// TwinCAT 3 PLC project haptix_beckhoff
// Title: Haptix-Beckhoff
// Company: HaptiX Lab
// Author: Nick Janne
// ProjectVersion: 0.5
// Description: This is a library containing a standardized set of function blocks and tools used in research projects at the HaptiX Lab at the University of Michigan
// ProgramVersion: 3.1.4024.0
// libraries:
//   Tc2_Standard, * (Beckhoff Automation GmbH)
//   Tc2_System, * (Beckhoff Automation GmbH)
//   Tc3_Module, * (Beckhoff Automation GmbH)
// project tree:
//   / PlcTask.TcTTO
//   POUs/ FB_AnalogLoadCellInput.TcPOU, FB_AnalogMotorDriver.TcPOU, FB_QuadratureEncoder.TcPOU, Test_AnalogInput.TcPOU, Test_AnalogMotorDriver.TcPOU
// real-time tasks:
//   TASK PlcTask: cycle T#10ms, priority 20, ADS port 350
// I/O:
//   DEVICE Device 2 (EtherCAT), AmsNetId 141.212.76.55.3.1
//     Term 1 (EK1100) [EK1100 EtherCAT Coupler (2A E-Bus)]
//       Term 2 (EL4038) [EL4038 8Ch. Ana. Output +/-10V, 12bit]
//       Term 3 (EL3174) [EL3174 4Ch. Ana. Input +/-10V Diff., +/-20mA SingleEnded, 16 Bit]
//       Term 4 (EL5122) [EL5122 2Ch. Inc. Encoder 5V (2xAB TTL)]
//       Term 5 (EL9011) [EL9011 End Terminal]
// variable links:
//   haptix-beckhoff/haptix-beckhoff Instance <-> Device 2 (EtherCAT)/Term 1 (EK1100)/Term 3 (EL3174)
//     PlcTask Inputs/Test_AnalogInput.fbLoadCell.nAnalogReading <-> AI Standard Channel 1/Value

CONFIGURATION haptix_beckhoff
    RESOURCE PLC ON TwinCAT3
        TASK PlcTask(INTERVAL := T#10ms, PRIORITY := 20);
        PROGRAM Test_AnalogInput WITH PlcTask : Test_AnalogInput;
    END_RESOURCE
END_CONFIGURATION

// ---- POUs/Test_AnalogInput.TcPOU
PROGRAM Test_AnalogInput
VAR
	fbLoadCell : FB_AnalogLoadCellInput; 
	rOutputNewtons : REAL; 
END_VAR

fbLoadCell(); 
rOutputNewtons := fbLoadCell.rCalibratedOutput;

END_PROGRAM

// ---- POUs/FB_AnalogLoadCellInput.TcPOU
FUNCTION_BLOCK FB_AnalogLoadCellInput
VAR_INPUT
	rYIntercept : REAL := -72.1; // Y intercept when fitting a line for Integer Counts (Y) v.s. Applied Mass (X) 
	rXSlope : REAL := -371; // Slope when fitting a line for Integer Coutns (Y) v.s. Applied Mass (X)
	sUnits : STRING := 'N'; 
END_VAR
VAR_OUTPUT
	nRawCounts : INT; // Copied from nAnalogReading
	rCalibratedOutput : REAL; 
	sOutputUnits : STRING; // Copied from sUnits 
END_VAR
VAR
	nAnalogReading AT %I* : INT; 
END_VAR

// First get the analog reading, and save it 
nRawCounts := nAnalogReading; 

// Then, convert the reading to get the output in calibrated format: 
rCalibratedOutput := (nRawCounts - rYIntercept) * (1/(rXSlope)); 

// Finally, copy over the units 
sOutputUnits := sUnits;

END_FUNCTION_BLOCK

// ---- POUs/FB_AnalogMotorDriver.TcPOU
FUNCTION_BLOCK FB_AnalogMotorDriver
VAR_INPUT
	// Nominally, respect requested command voltage between (-10)-10V, i.e. if rCommandVoltage
	// is 5, then the output on the channel should be 5V. However, we can alternatively 
	// Request voltage in normalized mode, which considers rCommandVoltage as a 
	// normalized signal between (-1)-1. To enable this mode, set the bUseNormalizedScale
	// flag, which is defaulted to false. When normalized signals are used, the user can additionally 
	// specify whether normalized commands map to (-10)-10V, or (-5)-5V; the latter is triggered
	// when bUseHalfScale is set to TRUE. 
	rCommandVoltage : REAL;
	bUseNormalizedScale : BOOL := FALSE;
	bUseHalfScale : BOOL := FALSE; 
END_VAR
VAR_OUTPUT
	nPosAnalogOutput AT %Q* : INT; 
	nNegAnalogOutput AT %Q* : INT; 
	nZeroRefAnalogOutput AT %Q* : INT;
	rActualCommandVoltage : REAL;  
	bOutputInError : BOOL; 
END_VAR
VAR
	nTEN_VOLT_AMPLITUDE : INT := 32767; 
	nFIVE_VOLT_AMPLITUDE : INT := 16383;
END_VAR

IF bUseNormalizedScale THEN
	
	// Again check if argument is valid
	IF ABS(rCommandVoltage) > 1 THEN 
		bOutputInError := TRUE; 
		RETURN;
	END_IF
	
	// Check to see if we should use the half scale. 
	IF bUseHalfScale THEN
		nPosAnalogOutput := REAL_TO_INT(rCommandVoltage * nFIVE_VOLT_AMPLITUDE); 
		rActualCommandVoltage := rCommandVoltage * 5.0; 
	ELSE
		nPosAnalogOutput := REAL_TO_INT(rCommandVoltage * nTEN_VOLT_AMPLITUDE);
		rActualCommandVoltage := rCommandVoltage * 10.0;  
	END_IF
	
	nNegAnalogOutput := -1 * nPosAnalogOutput;  
	bOutputInError := FALSE; 
	
ELSE 
	// In this case we were passed a raw voltage signal. 
	// Should check to see if scaling is appropriate, etc. 
	IF ABS(rCommandVoltage) > 10 THEN
		bOutputInError := TRUE; 
		RETURN; 
	END_IF
	
	rActualCommandVoltage := rCommandVoltage;
	nPosAnalogOutput := REAL_TO_INT(rCommandVoltage * nTEN_VOLT_AMPLITUDE / 10.0);
	nNegAnalogOutput := -1 * nPosAnalogOutput;  
	
	bOutputInError := FALSE;
	
END_IF

METHOD Reset : BOOL
VAR_INPUT
END_VAR
nPosAnalogOutput := 0; 
nNegAnalogOutput := 0; 
nZeroRefAnalogOutput := 0; 
bOutputInError := FALSE;
END_METHOD

END_FUNCTION_BLOCK

// ---- POUs/FB_QuadratureEncoder.TcPOU
FUNCTION_BLOCK FB_QuadratureEncoder
VAR_INPUT
	nCPR : UINT := 2048; // Counts per revolution of encoder
END_VAR
VAR_OUTPUT
	rDegrees : REAL := 0; 
	rLastDegrees : REAL := 0; 
	rRadians : REAL := 0; 
	rLastRadians : REAL := 0; 
	nNetCounts : LINT := 0; 
END_VAR
VAR	
	// This is a single channel of a two-channel quadrature encoder 
	// (if using the EL5122). This QE_CHANNEL object maps all the data
	// we want directly (counts) FROM the device manager 
	// found in the IO tab TO this quadrature encoder block right here. 
	// The quadrature encoder block abstracts any complexity needed 
	// to read/set values in the QE_CHANNEL object so that the device 
	// works as seemlessly as possible. 
	QE_CHANNEL_COUNTS AT %I* : UDINT; 	
	
	// We also create some additional variables to keep track of things 
	// for degrees calculation 
	nMAX_ENCODER_COUNT : ULINT := 16#100000000; // 2^32
	bLastCountInitialized : BOOL := FALSE; 
	nLastCount : UDINT; 
	
END_VAR

// Here, we first check to see if initialized, and then 
// we update the position value. 
IF NOT bLastCountInitialized THEN 
	nLastCount := QE_CHANNEL_COUNTS;
	bLastCountInitialized := TRUE; 
END_IF

// First we call a function to update the cumulated counts value 
UpdateNetCounts();

// Then we convert to degrees as well as updating last degrees 
UpdateDegrees(); 
UpdateRadians();

METHOD Reset : BOOL
VAR_INPUT
END_VAR
bLastCountInitialized := FALSE; 
nNetCounts := 0; 
rDegrees := 0;
END_METHOD

METHOD UpdateDegrees : BOOL
VAR_INPUT
END_VAR
// Here, we simply take the current net counts value 
// and convert it to degrees. We also take note 
// of the previous degrees value and store in last degrees
rLastDegrees := rDegrees; 
rDegrees := LINT_TO_REAL(nNetCounts) * 360.0 / (4 * nCPR); 
UpdateDegrees := TRUE;
END_METHOD

METHOD UpdateNetCounts : BOOL
VAR_INPUT
END_VAR
VAR
	nCurrentCount : UDINT; 
	nForwardDistance : ULINT; 
	nBackwardDistance : ULINT; 
END_VAR
// First get the current coutns 
nCurrentCount := QE_CHANNEL_COUNTS; 

// Quickly check if we can exit early
IF nCurrentCount = nLastCount THEN 
	UpdateNetCounts := TRUE; 
	RETURN; 
END_IF

// Otherwise, calculate forward, backward distances 
nForwardDistance := (nCurrentCount - nLastCount + nMAX_ENCODER_COUNT) MOD nMAX_ENCODER_COUNT; 
nBackwardDistance := (nLastCount - nCurrentCount + nMAX_ENCODER_COUNT) MOD nMAX_ENCODER_COUNT; 

IF nForwardDistance <= nBackwardDistance THEN 
	nNetCounts := nNetCounts + ULINT_TO_LINT(nForwardDistance); 
ELSIF nBackwardDistance < nForwardDistance THEN 
	nNetCounts := nNetCounts - ULINT_TO_LINT(nBackwardDistance); 
ELSE 
	UpdateNetCounts := FALSE; // Error has occured 
	RETURN; 
END_IF

nLastCount := nCurrentCount; 
UpdateNetCounts := TRUE;
END_METHOD

METHOD UpdateRadians : BOOL
VAR_INPUT
END_VAR
// Here, we simple take the current net counts value 
// and convert it to radians. We also take note 
// of the previous radians value and store in last radians
rLastRadians := rRadians; 
rRadians := LINT_TO_REAL(nNetCounts) * 2 * PI / (4 * nCPR); 
UpdateRadians := TRUE;
END_METHOD

END_FUNCTION_BLOCK

// ---- POUs/Test_AnalogMotorDriver.TcPOU
PROGRAM Test_AnalogMotorDriver
VAR
	AM_Driver : FB_AnalogMotorDriver; 
	fbSystemTime : GETSYSTEMTIME; 
	lowerHalf : UDINT; // Lower 32 bits 
	upperHalf : UDINT; // Upper 32 bits 
	fullTime : ULINT; // Combined 64 bits
	currentTimeSeconds : LREAL; 
	elapsedSeconds : LREAL; 
	
	bInitialTimeSet : BOOL := FALSE; 
	initialTimeSeconds : LREAL; // To store initial time for reference 
	
	// Output values for sine 
	rSineSignal : LREAL; 
	nPosOutputCommand : INT; 
	nNegOutputCommand : INT; 
	
END_VAR

// Poll the current system time 
fbSystemTime();
lowerHalf := fbSystemTime.timeLoDW; 
upperHalf := fbSystemTime.timeHiDW; 

fullTime := SHL(UDINT_TO_ULINT(upperHalf), 32) OR UDINT_TO_ULINT(lowerHalf); 
currentTimeSeconds := ULINT_TO_LREAL(fullTime) / 10000000.0; 

// Check to see if we need to set our initial condition. 
IF NOT bInitialTimeSet THEN
	initialTimeSeconds := currentTimeSeconds; 
	bInitialTimeSet := TRUE; 
END_IF

// Then get the DT 
elapsedSeconds := currentTimeSeconds - initialTimeSeconds; 

// Finally, pass the sine value to see what's up 
rSineSignal := 2 * SIN(elapsedSeconds * 2 * 3.14); 
AM_Driver(rCommandVoltage := rSineSignal); 
nPosOutputCommand := AM_Driver.nPosAnalogOutput; 
nNegOutputCommand := AM_Driver.nNegAnalogOutput;

END_PROGRAM
